FUNCTION_BLOCK FB_ItemRegister
VAR_INPUT
	bSignal					: BOOL;
	bReset					: BOOL;
END_VAR
VAR_OUTPUT
	aItemOnTimeRegistry		: ARRAY[0..GVL_Constant.ITEM_ARRAY_SIZE] OF TIME;
	aItemOffTimeRegistry	: ARRAY[0..GVL_Constant.ITEM_ARRAY_SIZE] OF TIME;
	
	nTimeCount				: INT;
END_VAR
VAR
	tTimeOn					: TON;
	tReadTimeOn				: TIME;
	osReadOnTime			: F_TRIG;
	
	tTimeOFF				: TON;
	tReadTimeOff			: TIME;
	osReadOffTime			: R_TRIG;
	
	i						: INT;
END_VAR

IF bSignal THEN
	tTimeOn(IN:=TRUE, PT:=T#5S, ET=>tReadTimeOn);
ELSE
	tTimeOFF(IN:=TRUE, PT:=T#5S, ET=>tReadTimeOff);
END_IF;

//Write on time to array
M_ReadOnTime();

//Write off time to array
M_ReadOffTime();

//Reset array for time registry
M_ResetTimeRegistry();

//On R_Trig of Signal
METHOD PUBLIC M_ReadOffTime
VAR_INPUT
END_VAR
osReadOffTime(CLK:=bSignal);

IF osReadOffTime.Q THEN
	aItemOffTimeRegistry[nTimeCount] := tReadTimeOff;
	tTimeOff(IN:=FALSE);
END_IF
END_METHOD

//On F_Trig of Signal
METHOD PUBLIC M_ReadOnTime
VAR_INPUT
END_VAR
VAR
END_VAR
osReadOnTime(CLK:=bSignal);

IF osReadOnTime.Q THEN
	aItemOnTimeRegistry[nTimeCount] := tReadTimeOn;
	nTimeCount := nTimeCount +1;
	tTimeOn(IN:=FALSE);
END_IF
END_METHOD

METHOD PUBLIC M_ResetTimeRegistry
VAR_INPUT
END_VAR
IF bReset THEN
	tTimeOFF(IN:=FALSE);
	tTimeOn(IN:=FALSE);
	
	FOR i := 0 TO nTimeCount DO 
		aItemOffTimeRegistry[i] := T#0S;
		aItemOnTimeRegistry [i] := T#0S;
	END_FOR
	
	nTimeCount := 0;	
	bReset := FALSE;
END_IF
END_METHOD

END_FUNCTION_BLOCK

(* stored: Version 1.1.0.1, ProductVersion 3.1.4024.12
   POU FB_ItemRegister: Id {c0a9bbfd-92cb-44d8-9279-e542f10353df}, SpecialFunc None
   Method M_ReadOffTime: Id {0dd02e9a-9bb9-495a-8635-92fa2193c059}
   Method M_ReadOnTime: Id {5f071343-b7ea-4d4c-8e55-b7e89db6d0ee}
   Method M_ResetTimeRegistry: Id {aec981ff-8120-4b14-9fab-616a1f61d830} *)
